PROGRAM MAIN
VAR
	RunnerTests : RunnerTestSuite;
	ObjectTests : ObjectTestSuite;
END_VAR

RunnerTests();
ObjectTests();

END_PROGRAM

(* stored: Version 1.1.0.1
   POU MAIN: Id {45608e08-666f-403e-a083-2e21d622d99c}, SpecialFunc None *)
